FUNCTION_BLOCK FB_CB_AuxMVCB EXTENDS FB_CB_Base
//////////////////
//  Motorized Circuit Breaker with telecommAND   Requires Open and Close impulsions.
//////////////////

VAR_INPUT PERSISTENT
	// Parameters of the Object (instance/model specific) 
	ParamTP_Impulsion	   : TIME := T#2S;			(* (s)  Config : Tempo for the start or stop command impulsion*)
	ParamFuseNC		       : BOOL;					(* (NA) False: TRUE = Closed , True : TRUE = opened	*)
END_VAR

VAR_OUTPUT
	//Child objects
	
END_VAR

VAR_INPUT
	// I/O Inputs              
	IN_MesFuse_IO			: BOOL;
	IN_MesEarth_IO			: BOOL; 
	
END_VAR

VAR
	//M_OPENCLOSE VARIABLES//	
		RsFuse				:RS;
		
	//M_ALARMMANAGEMENT VARIABLES//
	MesDataExd	: CB_AuxMVCB_Sch;
 
	//M_STATEMANAGER VARIABLES//
	
	// M_EXECUTE VARIABLES //
		
 
END_VAR

METHOD M_AlarmManagement
//////////////////
// Manages Contactor alarms and warnings
/////////////////

VAR 
	// Method local variables (reinitialized at each cycle) 
	FB_AlarmCodeManager			: FB_AlarmCodeManager ; 	
END_VAR
// Check if command and measures are matching after tempo

TON_NotClosedAndNotOpened(IN:=  NOT MesClosed AND NOT MesOpened , PT := ParamTimeOut_Alarm) ; 
TON_ClosedAndOpened(IN:=MesClosed AND MesOpened, PT := ParamTimeOut_Alarm) ; 

RsFuse(Set:= MesDataExd.MesFuseBurned ,Reset1:=GVL_CFG.CmdClearFault_G OR IN_CmdReset_L);

// ALARM CODE //
	FB_AlarmCodeManager(
		bAlarm1			:= FALSE,										//
		bAlarm2			:= TON_NotClosedAndNotOpened.Q,					// Incoherent state mesure (neither open nor closed) 
		bAlarm3 		:= TON_ClosedAndOpened.Q, 						// Incoherent state mesure (Open and closed)	
		bAlarm4			:= RsFuse.Q1,									// Fuse is burned
		bAlarm5			:= FALSE, 										//  
		bAlarm6			:= FALSE, 										//
		bAlarm7			:= FALSE,                                       //
		bAlarm8			:= FALSE,                                       //
		bAlarm9			:= FALSE,                                       //
		bAlarm10		:= FALSE,                                       //
		bAlarm11		:= FALSE,                                       //
		bAlarm12		:= FALSE,                                       //
		bAlarm13		:= FALSE, 										//
		bAlarm14		:= FALSE, 										//
		bAlarm15		:= FALSE , 										// 
		wAlarmCode		=>MesDataExd.MesData.MesAlarmCode);

//WARNING CODE//
		FB_AlarmCodeManager(
		bAlarm1			:= FALSE, 										// 
		bAlarm2			:= FALSE,	 									// 
		bAlarm3 		:= FALSE,										// 
		bAlarm4			:= FALSE, 										// 
		bAlarm5			:= FALSE, 										//
		bAlarm6			:= MesDataExd.MesEarth, 						// Earthing mode
		bAlarm7			:= FALSE, 										//
		bAlarm8			:= FALSE,                                       //
		bAlarm9			:= FALSE,                                       //
		bAlarm10		:= FALSE,                                       //
		bAlarm11		:= FALSE,                                       //
		bAlarm12		:= FALSE,                                       //
		bAlarm13		:= FALSE,                                       //
		bAlarm14		:= FALSE,                                       //
		bAlarm15		:= FALSE, 										//
		wAlarmCode 		=>MesDataExd.MesData.MesWarningCode);

// EVENT CODE //
	FB_AlarmCodeManager(
		bAlarm1			:= FALSE, 										// 
		bAlarm2			:= FALSE, 										// 
		bAlarm3			:= MesOpened, 									// Open position
		bAlarm4			:= MesClosed, 									// Closed position
		bAlarm5			:= IN_CmdReset_L, 								// Reset Command
		bAlarm6			:= FALSE, 										//
		bAlarm7			:= FALSE,                                       //
		bAlarm8			:= FALSE,                                       //
		bAlarm9			:= FALSE,                                       //
		bAlarm10		:= FALSE,                                       //
		bAlarm11		:= FALSE,                                       //
		bAlarm12		:= FALSE,                                       //
		bAlarm13		:= FALSE,                                       //
		bAlarm14		:= FALSE, 										//
		bAlarm15		:= FALSE, 										//
		wAlarmCode		=>MesDataExd.MesData.MesEventCode);
		
	// UPDATE STRUCTURE


	IF NOT ParamFuseNC THEN 
	MesDataExd.MesFuseBurned := NOT IN_MesFuse_IO;
	ELSE
	MesDataExd.MesFuseBurned := IN_MesFuse_IO;
	END_IF
MesDataExd.MesEarth	:= IN_MesEarth_IO ;
END_METHOD

METHOD M_Execute
VAR_INPUT
END_VAR
// PERMANENT CONDITIONS //	
MesDataExd.MesData.MesCP_Open					:= IN_CmdOpen AND NOT IN_CmdReset_L;
MesDataExd.MesData.MesCP_Close				:= NOT MesDataExd.MesData.MesClosed AND IN_CmdClose AND NOT MesDataExd.MesData.MesAlarmCode.0 AND NOT MesDataExd.MesData.MesCP_Open AND NOT IN_CmdReset_L ;


SUPER^.M_Execute();
END_METHOD

METHOD M_OpenClose
//////////////////
// Manages Opening and Closing of the contactor
//////////////////

VAR 
	// Method local variables (reinitialized at each cycle) 

	
END_VAR
END_METHOD

METHOD M_StateManager
//////////////////
// Manages Contactor State
/////////////////

VAR 
	// Method local variables (reinitialized at each cycle) 
	
END_VAR
MesState := 0 ; 
IF MesOpened THEN		// If the cell seems opens and closed in the same time, we will consider it as opened. 
	
	MesState.0 := 1 ; 
MesDataExd.MesData.MesClosed := FALSE ; 
MesDataExd.MesData.MesOpened := TRUE ; 
ELSIF MesClosed THEN
	
	MesState.1 := 1 ; 
MesDataExd.MesData.MesClosed := TRUE ; 
MesDataExd.MesData.MesOpened := FALSE ; 
ELSE 
	MesState.0 := 1 ;		// if the cell seems neither opened and neither closed , we will consider it as opened. 
MesDataExd.MesData.MesClosed := FALSE ; 	
MesDataExd.MesData.MesOpened := TRUE ; 
END_IF
END_METHOD

END_FUNCTION_BLOCK

(* stored: Version 1.1.0.1, ProductVersion 3.1.4024.6
   POU FB_CB_AuxMVCB: Id {5254a75b-1653-4817-88d3-f422ce31f957}, SpecialFunc None
   Method M_AlarmManagement: Id {58a40b5e-bb95-4fa1-b6b1-b619b9b836aa}
   Method M_Execute: Id {8c338fdd-d981-492a-bf9e-371e6f5f0f63}
   Method M_OpenClose: Id {b49bddbb-67c6-402f-87b6-86436312f4d7}
   Method M_StateManager: Id {091e174f-72e5-4698-bef0-aeaf41cb2310} *)
